// Mitsubishi GX Works2 project: WheelValveDrillFX3S   PLC: FX3S

// global labels: Global1
VAR_GLOBAL
  Run AT M1 : BOOL;
  RunStop AT M2 : BOOL;
  RunState AT D0 : INT;
  AccelTime AT D1 : INT;
  DecelTime AT D2 : INT;
  XXBusy AT M8340 : BOOL;
  XXPos AT D8340 : DINT;
  XXAccelTime AT D8348 : INT;
  XXDecelTime AT D8349 : INT;
  XXPosView AT D3 : DINT;
  XXTarPos AT D5 : DINT;
  XXFeed AT D7 : DINT;
  XXTarR AT M4 : BOOL;
  XXTarRSkip AT D9 : INT;
  XXOPulse AT Y000 : BOOL;
  XXODirection AT Y004 : BOOL;
  XXRun AT M7 : BOOL;
  XXDirection AT M8 : BOOL;
  RunI AT X000 : BOOL;
  XXMinI AT X002 : BOOL;
  XXMaxI AT X003 : BOOL;
  TapI AT X001 : BOOL;
  ClampO AT Y003 : BOOL;
  Clamp AT M10 : BOOL;
END_VAR

// task Task_01 (event TRUE, interval 0, priority 31): POU_01

PROGRAM POU_01
VAR
  fTmp : BOOL;
  fRunStateNext : BOOL;
  fRunStart : BOOL;
  fTapRise : BOOL;
END_VAR
MOV(M8002, 200, AccelTime);

SET(M8000 AND Run AND M100, fTmp);
RST(fTmp, Run);
MOV(fTmp, 1, RunState);
RST(fTmp, XXRun);
RST(fTmp, fTmp);

SET(fRunStart, fTmp);
RST(fTmp, fRunStart);
MOV(fTmp, 30, RunState);
RST(fTmp, XXRun);
RST(fTmp, Run);
RST(fTmp, fTmp);

SET(RunStop, fTmp);
RST(fTmp, RunStop);
MOV(fTmp, 30, RunState);
RST(fTmp, XXRun);
RST(fTmp, Run);
RST(fTmp, fTmp);

INC(fRunStateNext, RunState); RST(fRunStateNext, fRunStateNext);
DECO(TRUE, RunState, 6, M100);
DECO(TRUE, RunState, 6, M200); ZRST(NOT XXTarR, M200, M263);

(**)
(*not at min, move up*)
SET(M201 AND NOT XXMinI, fTmp);
RST(fTmp, XXPos);
DMOV(fTmp, -10000, XXTarPos);
DMOV(fTmp, 10000, XXFeed);
SET(fTmp, XXRun);
SET(fTmp, fRunStateNext); RST(fTmp, fTmp);
(*at min, not move up*)
SET(M201 AND XXMinI, fTmp);
MOV(fTmp, 3, RunState); RST(fTmp, fTmp);
(*move up done, stop*)
SET(M102 AND XXMinI, fTmp);
RST(fTmp, XXRun);
SET(fTmp, fRunStateNext); RST(fTmp, fTmp);
(*move down fast*)
SET(M203, fTmp);
RST(fTmp, XXPos);
SET(fTmp, Clamp);
DMOV(fTmp, 3000, XXTarPos);
DMOV(fTmp, 10000, XXFeed);
SET(fTmp, XXRun);
SET(fTmp, fRunStateNext); RST(fTmp, fTmp);
(*move down slow*)
SET(M204, fTmp);
DMOV(fTmp, 10000, XXTarPos);
DMOV(fTmp, 1500, XXFeed);
SET(fTmp, XXRun);
SET(fTmp, fRunStateNext); RST(fTmp, fTmp);
(*at max, stop*)
SET(M105 AND XXMaxI, fTmp);
RST(fTmp, XXRun);
SET(fTmp, fRunStateNext); RST(fTmp, fTmp);
(*move up fast*)
SET(M206, fTmp);
RST(fTmp, XXPos);
DMOV(fTmp, -10000, XXTarPos);
DMOV(fTmp, 10000, XXFeed);
SET(fTmp, XXRun);
SET(fTmp, fRunStateNext); RST(fTmp, fTmp);
(*move up done, stop*)
SET(M107 AND XXMinI, fTmp);
RST(fTmp, XXRun);
RST(fTmp, Clamp);
RST(fTmp, RunState);
RST(fTmp, fTmp);
(**)

(*start or stop rise, move up fast*)
SET(M230 AND NOT XXMinI, fTmp);
RST(fTmp, XXPos);
DMOV(fTmp, -10000, XXTarPos);
DMOV(fTmp, 10000, XXFeed);
SET(fTmp, XXRun);
SET(fTmp, fRunStateNext); RST(fTmp, fTmp);
(*at min, not move up*)
SET(M230 AND XXMinI, fTmp);
SET(fTmp, fRunStateNext); RST(fTmp, fTmp);
(*move up done, stop*)
SET(M131 AND XXMinI, fTmp);
RST(fTmp, XXRun);
RST(fTmp, RunState);
RST(fTmp, Clamp);
RST(fTmp, fTmp);

(*XX*)
RST(XXRun AND XXTarPos = XXPos, XXRun);
DDRVA(XXRun, XXTarPos, XXFeed, XXOPulse, XXODirection);
RST(M8029, XXRun);
OUT(XXODirection, XXDirection);
INC(NOT XXRun AND NOT XXBusy AND XXTarRSkip < 5, XXTarRSkip);
RST(XXRun, XXTarRSkip);
OUT(XXTarRSkip >= 5, XXTarR);

(*Input*)
PLS(RunI, fRunStart); SET(fRunStart, fRunStart);
PLF(RunI, RunStop); SET(RunStop, RunStop);
PLS(TapI, fTapRise); SET(fTapRise AND RunI, Run);

(*Output*)
OUT(Clamp, ClampO);
END_PROGRAM
